DATA_BLOCK "DB2000_ED"
TITLE = DB2000_ED
{ S7_Optimized_Access := 'FALSE' }
AUTHOR : HCR
FAMILY : ZeusControl
VERSION : 1.0
//Bloque de datos entrada digital
   STRUCT
      ED : Array[0.."N_MAX_DISP_ED"] of "UDT_ZC_DISP_ED";
      Mux { S7_SetPoint := 'False'} : Array[0.."N_MAX_MUX_DISP"] of "UDT_ZC_DISP_MUX_ED";
      Agrup : Array[0.."N_MAX_DISP_AGRUP"] of "UDT_ZC_DISP_AGRUP";
   END_STRUCT;


BEGIN
   ED[0].Hmi_Estado := 0;
   ED[0].Estado_AutoMan := FALSE;
   ED[0].Estado_Activado := FALSE;
   ED[0].Estado_EntradaCanal := FALSE;
   ED[0].Orden_ActivarManual := FALSE;
   ED[0].Config_Habilitar := FALSE;
   ED[0].Config_HabilitarRetardoAct := FALSE;
   ED[0].Config_HabilitarRetardoDes := FALSE;
   ED[0].Config_HabilitarInvertir := FALSE;
   ED[0].Aux_oldActivado := FALSE;
   ED[0].Aux_oldAutoMan := FALSE;
   ED[0].Config_GrupoAlarma := 0;
   ED[0].Config_DireccionEntradaByte := 0;
   ED[0].Config_DireccionEntradaBit := 0;
   ED[0].Tiempos_SetPointTiempoAct := 3;
   ED[0].Tiempos_SetPointTiempoDes := 3;
   ED[0].Tiempos_TiempoAct := 0;
   ED[0].Tiempos_TiempoDes := 0;
   ED[1].Hmi_Estado := 1;
   ED[1].Estado_AutoMan := FALSE;
   ED[1].Estado_Activado := FALSE;
   ED[1].Estado_EntradaCanal := FALSE;
   ED[1].Orden_ActivarManual := FALSE;
   ED[1].Config_Habilitar := TRUE;
   ED[1].Config_HabilitarRetardoAct := FALSE;
   ED[1].Config_HabilitarRetardoDes := FALSE;
   ED[1].Config_HabilitarInvertir := FALSE;
   ED[1].Aux_oldActivado := FALSE;
   ED[1].Aux_oldAutoMan := FALSE;
   ED[1].Config_GrupoAlarma := 0;
   ED[1].Config_DireccionEntradaByte := 112;
   ED[1].Config_DireccionEntradaBit := 6;
   ED[1].Tiempos_SetPointTiempoAct := 8;
   ED[1].Tiempos_SetPointTiempoDes := 7;
   ED[1].Tiempos_TiempoAct := 0;
   ED[1].Tiempos_TiempoDes := 0;
   Mux[0].Habilitar := TRUE;
   Mux[0].ExisteCambio := FALSE;
   Mux[0].MaxVisible := FALSE;
   Mux[0].Index := 53;
   Mux[0].oldIndex := 53;
   Mux[0].ED.Hmi_Estado := 9;
   Mux[0].ED.Estado_AutoMan := FALSE;
   Mux[0].ED.Estado_Activado := TRUE;
   Mux[0].ED.Estado_EntradaCanal := TRUE;
   Mux[0].ED.Orden_ActivarManual := TRUE;
   Mux[0].ED.Config_Habilitar := TRUE;
   Mux[0].ED.Config_HabilitarRetardoAct := FALSE;
   Mux[0].ED.Config_HabilitarRetardoDes := FALSE;
   Mux[0].ED.Config_HabilitarInvertir := FALSE;
   Mux[0].ED.Aux_oldActivado := TRUE;
   Mux[0].ED.Aux_oldAutoMan := FALSE;
   Mux[0].ED.Config_GrupoAlarma := 1;
   Mux[0].ED.Config_DireccionEntradaByte := 205;
   Mux[0].ED.Config_DireccionEntradaBit := 4;
   Mux[0].ED.Tiempos_SetPointTiempoAct := 3;
   Mux[0].ED.Tiempos_SetPointTiempoDes := 3;
   Mux[0].ED.Tiempos_TiempoAct := 0;
   Mux[0].ED.Tiempos_TiempoDes := 0;
   Mux[1].Habilitar := TRUE;
   Mux[1].ExisteCambio := FALSE;
   Mux[1].MaxVisible := FALSE;
   Mux[1].Index := 0;
   Mux[1].oldIndex := 0;
   Mux[1].ED.Hmi_Estado := 0;
   Mux[1].ED.Estado_AutoMan := FALSE;
   Mux[1].ED.Estado_Activado := FALSE;
   Mux[1].ED.Estado_EntradaCanal := FALSE;
   Mux[1].ED.Orden_ActivarManual := FALSE;
   Mux[1].ED.Config_Habilitar := FALSE;
   Mux[1].ED.Config_HabilitarRetardoAct := FALSE;
   Mux[1].ED.Config_HabilitarRetardoDes := FALSE;
   Mux[1].ED.Config_HabilitarInvertir := FALSE;
   Mux[1].ED.Aux_oldActivado := FALSE;
   Mux[1].ED.Aux_oldAutoMan := FALSE;
   Mux[1].ED.Config_GrupoAlarma := 0;
   Mux[1].ED.Config_DireccionEntradaByte := 0;
   Mux[1].ED.Config_DireccionEntradaBit := 0;
   Mux[1].ED.Tiempos_SetPointTiempoAct := 3;
   Mux[1].ED.Tiempos_SetPointTiempoDes := 3;
   Mux[1].ED.Tiempos_TiempoAct := 0;
   Mux[1].ED.Tiempos_TiempoDes := 0;
   Agrup[0].AlgunaEnManual := FALSE;
   Agrup[0].AlgunaAlarma := FALSE;
   Agrup[0].NuevaAlarma := FALSE;
   Agrup[1].AlgunaEnManual := FALSE;
   Agrup[1].AlgunaAlarma := FALSE;
   Agrup[1].NuevaAlarma := FALSE;

END_DATA_BLOCK

